DATA_BLOCK "AllPump_DB"   // DB9
VERSION : 0.1
// stored: AutoNumber true, DBAccessibleFromOPCUA true, InstanceOfName AllPump, InstanceOfType FB
"AllPump"
BEGIN
END_DATA_BLOCK

DATA_BLOCK "Sequencer_DB"   // DB17
VERSION : 0.1
// stored: AutoNumber true, DBAccessibleFromOPCUA true, InstanceOfName Sequencer, InstanceOfType FB
"Sequencer"
BEGIN
END_DATA_BLOCK

DATA_BLOCK "hardwareTimePulse_DB"   // DB18
VERSION : 0.1
// stored: AutoNumber true, DBAccessibleFromOPCUA true, InstanceOfName hardwareTimePulse, InstanceOfType FB
"hardwareTimePulse"
BEGIN
END_DATA_BLOCK

DATA_BLOCK "tmrAck"   // DB10
{ S7_Optimized_Access := 'TRUE' }
// stored: AutoNumber true, DBAccessibleFromOPCUA true, InstanceOfName IEC_TIMER, OfSystemLibElement IEC_TIMER, OfSystemLibVersion 1.0
"IEC_TIMER"
   // VAR
   //    PT : Time;
   //    ET { ExternalWritable := 'False'} : Time;
   //    IN : Bool;
   //    Q { ExternalWritable := 'False'} : Bool;
   // END_VAR
BEGIN
END_DATA_BLOCK

DATA_BLOCK "AllFlowCounter_DB"   // DB23
VERSION : 0.1
// stored: AutoNumber true, DBAccessibleFromOPCUA true, InstanceOfName AllFlowCounter, InstanceOfType FB
"AllFlowCounter"
   // VAR
   //    prewHour : USInt;
   //    prewDay : USInt;
   //    FM201 { S7_SetPoint := 'True'} : "VolumeCounter";
   //    FM501 { S7_SetPoint := 'True'} : "VolumeCounter";
   //    FM502 { S7_SetPoint := 'True'} : "VolumeCounter";
   //    FM901 { S7_SetPoint := 'True'} : "VolumeCounter";
   //    FM902 { S7_SetPoint := 'True'} : "VolumeCounter";
   //    FM1201 { S7_SetPoint := 'True'} : "VolumeCounter";
   //    FM1301 { S7_SetPoint := 'True'} : "VolumeCounter";
   //    FM1302 { S7_SetPoint := 'True'} : "VolumeCounter";
   //    FM1701 { S7_SetPoint := 'True'} : "VolumeCounter";
   //    FM1801 { S7_SetPoint := 'True'} : "VolumeCounter";
   // END_VAR
BEGIN
END_DATA_BLOCK

DATA_BLOCK "AllUF_DB"   // DB17
VERSION : 0.1
// stored: AutoNumber true, DBAccessibleFromOPCUA true, InstanceOfName AllUF, InstanceOfType FB
"AllUF"
BEGIN
END_DATA_BLOCK

DATA_BLOCK "AllUfParam_DB"   // DB22
VERSION : 0.1
// stored: AutoNumber true, DBAccessibleFromOPCUA true, InstanceOfName AllUfParam, InstanceOfType FB
"AllUfParam"
BEGIN
END_DATA_BLOCK
